METHOD testNotIsEqualTo
VAR_INPUT
	(* for the test it's the parameter ``address1`` *)
	address1	:PVOID;
	(* for the test it's the parameter ``address2`` *)
	address2	:PVOID;
END_VAR
VAR
	(* just the expectation if the assertion to test must be worng or true *)
	assertionIsWrong		:BOOL;
	(* contains the format string for the test message *)
	message					:Tc2_System.T_MaxString;
	(* TwinCAT printf with the test message *)
	messageStringBuilder	:Tc2_Utilities.FB_FormatString;
END_VAR
THIS^.assertorContainer.resetAssertor();

assertionIsWrong := (address1 = address2);
message := SEL(
	assertionIsWrong,
	'address1 is 16#%X address2 is 16#%X assertion must be TRUE', 
	'address1 is 16#%X address2 is 16#%X assertion must be FALSE'
);
messageStringBuilder(
	sFormat := message,
	arg1 := THIS^.AnyToArg(address1),
	arg2 := THIS^.AnyToArg(address2)
);

THIS^.assertorContainer.assertor.assert.pointers.isNotEqualTo(
	address1 := address1,
	address2 := address2,
	message := ''
);

THIS^.AssertEquals_BOOL(
	Expected 	:= assertionIsWrong,
	Actual 		:= THIS^.assertorContainer.wasAssertionWrong,
	Message 	:= messageStringBuilder.sOut
);
END_METHOD

END_FUNCTION_BLOCK

(* stored: Version 1.1.0.1, ProductVersion 3.1.4026.13
   POU PointerAssertionsTests: Id {f966415f-df04-4a32-8a29-16669983edb0}, SpecialFunc None
   Folder internal: Id {16a01329-6f8f-4715-8438-d07ad7e6161f}
   Folder isAligned: Id {688c8f52-5144-4aae-a077-1473cbf86e08}
   Folder isDwordAligned: Id {7e4a20cb-f4f3-4fb7-beba-476b17cc17b4}
   Folder isEqualTo: Id {f6a4cbf1-1207-400c-99f3-38a94c446efb}
   Folder isLwordAligned: Id {5f20fb66-0a16-47df-9bc9-9e780c0e5db0}
   Folder isNotEqualTo: Id {a76f4de4-418b-46ad-9551-2a2f68744474}
   Folder isNotNull: Id {73627d3c-6876-48c6-b7af-7c1e1daf0942}
   Folder isNotOverlapping: Id {7c53f483-5518-411e-ae3c-70571d09516a}
   Folder isNull: Id {604d06f0-4dea-4ec9-b145-281256ca6ab4}
   Folder isOverlapping: Id {f6b7e754-398a-4416-a74e-8d6d3425679f}
   Folder isValid: Id {f785936a-463a-4e46-bca8-36861bda4c93}
   Folder isWordAligned: Id {7ebd3bcf-5231-4aaa-903f-fdd86a400d6d}
   Folder memoryAreaIsCnc: Id {1bb6cf7e-554e-46f4-90a6-26133547b0ef}
   Folder memoryAreaIsDynamic: Id {750e0adf-6744-46d2-b1a1-2cc6f692575c}
   Folder memoryAreaIsNotCnc: Id {40777263-6112-44dc-934d-32a2b65a1248}
   Folder memoryAreaIsNotDynamic: Id {fa684f57-7343-401e-8aed-882ea90a09cd}
   Folder memoryAreaIsNotStatic: Id {4cd59dfe-7b75-45b3-9276-a3be6fba4123}
   Folder memoryAreaIsNotUnknwon: Id {6c5b8299-2fec-4da7-887f-fc80176e8fe2}
   Folder memoryAreaIsStatic: Id {da7f60f0-4a54-4af0-b56a-bfd12c528964}
   Folder memoryAreaIsUnknwon: Id {6ad6294c-941b-4393-9953-88dbead16455}
   Method FB_exit: Id {203b1e30-c834-457e-9f98-e6fa2d484222}
   Method FB_reinit: Id {1d8b88d2-ae53-4f73-892b-9f4114a239c3}
   Method getTestNameFor: Id {edd87b13-f3ad-45f5-8400-b2f842dc34b7}
   Method init: Id {5081676b-37ce-409c-9cdd-a95d75abc2b2}
   Method leave: Id {f9313cde-9eb9-405d-b95c-ef4f2470faf0}
   Method memoryAreaToString: Id {e825c5cc-8329-4502-bb5f-f952316a7745}
   Method runIsAlignedTests: Id {273ccfb7-aacb-4c79-9c8d-e28908187a58}
   Method runIsDwordAlignedTests: Id {e19f25cc-1171-470b-bc0f-99f12cb67e17}
   Method runIsEqualToTests: Id {854ff968-96bd-478d-b06b-24df12472a0b}
   Method runIsLwordAlignedTests: Id {24633906-77ef-4ede-a287-6a11cc75355b}
   Method runIsNotEqualToTests: Id {0595c8c7-a657-41f3-a49b-4de819720503}
   Method runIsNotNullTests: Id {30fa128d-070e-4399-9697-d18e6e23344d}
   Method runIsNotOverlappingTests: Id {6589b4f1-14ed-4bfa-8605-5d445ca793dd}
   Method runIsNullTests: Id {e4dcff5c-5914-494a-a6e3-3f0de7b5d2ad}
   Method runIsOverlappingTests: Id {321cdd78-b49f-4e39-b530-7a6e81c4298d}
   Method runIsValidTests: Id {dbad4a73-c145-4443-a585-9a206ec69651}
   Method runIsWordAlignedTests: Id {2aabfc16-0b91-4524-bf8f-6801d0c9724b}
   Method runMemoryAreaIsCncTests: Id {e8f74879-fcc3-45e1-a8a1-ad50845a806f}
   Method runMemoryAreaIsDynamicTests: Id {6efd5f43-33cb-415d-8294-7c8294400f8f}
   Method runMemoryAreaIsNotCncTests: Id {7b2f6fa1-535f-4715-bcdc-cb771e0882e2}
   Method runMemoryAreaIsNotDynamicTests: Id {97ad892c-6dfc-4d0e-8fc1-47115ee0e2d5}
   Method runMemoryAreaIsNotStaticTests: Id {74ad6a09-71bd-4b50-b84b-22df99df5048}
   Method runMemoryAreaIsNotUnknownTests: Id {4168dbef-5670-418c-9d5e-7b43659982fe}
   Method runMemoryAreaIsStaticTests: Id {477331cc-9d86-46be-878b-3a0f4ddd257d}
   Method runMemoryAreaIsUnknownTests: Id {e77b08b1-9891-4ece-af7b-db9c4b7bd3c2}
   Method testIsAligned: Id {7c66c752-2040-4798-9203-b4a3e2fc686b}
   Method testIsDwordAligned: Id {89ca123f-e7e7-4011-9fd3-edfc3c0a67fc}
   Method testIsEqualTo: Id {f1b6fba6-3f19-4c60-b7e3-969319878ad0}
   Method testIsLwordAligned: Id {c2ff7d73-7a7a-4bba-aa0a-47440eac24fc}
   Method testIsNotNull: Id {020d7de3-0269-41e3-ad10-72fc760745b2}
   Method testIsNotOverlapping: Id {875b193c-a7bf-4d71-b27d-660c7d784bf4}
   Method testIsNull: Id {228b3f4a-1bea-4d6a-a686-67ef4262b8e5}
   Method testIsOverlapping: Id {dbfcfa33-4e1a-47ab-8a0e-d3e3005eebf7}
   Method testIsValid: Id {9c422e2f-ac8b-485c-89e5-893cda8483d2}
   Method testIsWordAligned: Id {b33fe127-0e45-4dab-a6ae-5a4879cbab3c}
   Method testMemoryAreaIsCnc: Id {d238ec4f-866d-42d3-b252-e9d37c9e8e55}
   Method testMemoryAreaIsDynamic: Id {fa5e2dc9-9546-43f0-b75d-96bf4024a4c8}
   Method testMemoryAreaIsNotCnc: Id {d92129d3-03b1-47f9-a5ce-c18024cb8bb4}
   Method testMemoryAreaIsNotDynamic: Id {ef2d64e5-a5b3-4e04-ad76-e61c89257f1d}
   Method testMemoryAreaIsNotStatic: Id {ce89fe5c-47b0-40f0-bf18-b26d579556d6}
   Method testMemoryAreaIsNotUnknown: Id {b9b832c9-aa2f-49c3-bea3-572608f1f351}
   Method testMemoryAreaIsStatic: Id {c22a8dde-5d04-42fd-9b34-a5a20788e2f6}
   Method testMemoryAreaIsUnknown: Id {29a5b5bb-3d05-47b8-bda7-93aebb3ef288}
   Method testNotIsEqualTo: Id {7ed70e97-990e-4e80-97a1-ccaa2c77ee71} *)
